PROGRAM Signals
VAR
	fbTimer1: TON;
	fbTimer2: TON;
	FB_Blinker1: FB_Blinker;
END_VAR

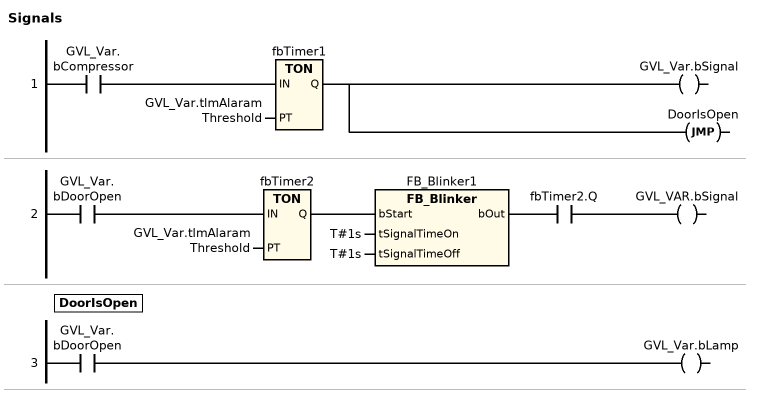
// NETWORK 1
fbTimer1(IN := GVL_Var.bCompressor, PT := GVL_Var.tlmAlaramThreshold); // TON
GVL_Var.bSignal := fbTimer1.Q;
IF fbTimer1.Q THEN JMP DoorIsOpen; END_IF

// NETWORK 2
fbTimer2(IN := GVL_Var.bDoorOpen, PT := GVL_Var.tlmAlaramThreshold); // TON
FB_Blinker1(bStart := fbTimer2.Q, tSignalTimeOn := T#1s, tSignalTimeOff := T#1s); // FB_Blinker
GVL_VAR.bSignal := FB_Blinker1.bOut AND fbTimer2.Q;

// NETWORK 3
DoorIsOpen:
GVL_Var.bLamp := GVL_Var.bDoorOpen;

END_PROGRAM

(* stored: Version 1.1.0.1, ProductVersion 3.1.4024.4
   POU Signals: Id {61bf3a1d-bcc9-489a-93a7-2ca13f8a54c5}, SpecialFunc None *)
